FUNCTION TryConvert_LWORD_TO_UDINT : BOOL
VAR_INPUT
	in : LWORD;
	out : REFERENCE TO UDINT;
END_VAR

IF in > DatatypeLimits.MAX_VALUE_OF_LWORD_WHICH_CAN_BE_HELD_IN_A_UDINT THEN
	RETURN;
END_IF

out := LWORD_TO_UDINT(in);
TryConvert_LWORD_TO_UDINT := TRUE;

END_FUNCTION

(* stored: Version 1.1.0.1, ProductVersion 3.1.4024.12
   POU TryConvert_LWORD_TO_UDINT: Id {85e584d7-a67a-4d16-a547-c4291aab47b5}, SpecialFunc None *)
